Staubli VAL3: io.dtx

public dio valve1 = {link=valve1}
public dio fIn0 = {link=fIn0}
public dio fIn1 = {link=fIn1}
public dio fOut0 = {link=fOut0}
